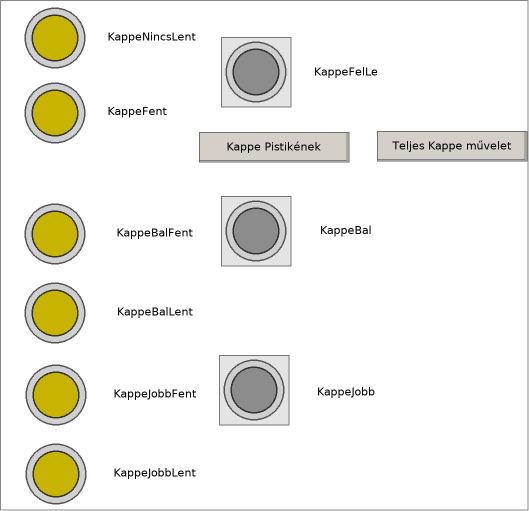
VISUALIZATION TempPistiKappe  // 529x511
    Group (20,3 187x70)
        Lamp1 (0,0 70x70), variable: GVL.bKappepresNincsLegalul, style: Lamp-Lamp1-Yellow
        Label (77,19 110x30), "KappeNincsLent"
    PushSwitch (221,37 70x70), variable: KAPPE.bKappeFelLe, behaviour: TOGGLE, style: Switch-PushSwitch-Gray
    Label (291,57 110x30), "KappeFelLe"
    Lamp1 (20,199 70x70), variable: KAPPE.bKappeBalFent, style: Lamp-Lamp1-Yellow
    Label (100,218 110x30), "KappeBalFent"
    Lamp1 (20,278 70x70), variable: KAPPE.bKappeBalLent, style: Lamp-Lamp1-Yellow
    Label (100,297 110x30), "KappeBalLent"
    PushSwitch (221,196 70x70), variable: KAPPE.bKappeBalFelLe, behaviour: TOGGLE, style: Switch-PushSwitch-Gray
    Label (291,216 110x29), "KappeBal"
    Lamp1 (21,360 70x70), variable: KAPPE.bKappeJobbFent, style: Lamp-Lamp1-Yellow
    Label (100,379 110x30), "KappeJobbFent"
    Lamp1 (21,439 70x70), variable: KAPPE.bKappeJobbLent, style: Lamp-Lamp1-Yellow
    Label (100,458 110x30), "KappeJobbLent"
    PushSwitch (219,355 70x70), variable: KAPPE.bKappeJobbFelLe, behaviour: TOGGLE, style: Switch-PushSwitch-Gray
    Label (291,377 110x30), "KappeJobb"
    Button (199,132 150x30), "Kappe Pistikének", input disabled if: KAPPE.bKappeBalFent<>KAPPE.bKappeJobbFent AND KAPPE.bKappeBalLent<>KAPPE.bKappeJobbLent
        OnMouseUp: execute {
            IF ((KAPPE.bKappeBalFent=TRUE) AND (KAPPE.bKappeBalLent=FALSE) AND (KAPPE.bKappeJobbFent=TRUE) AND (KAPPE.bKappeJobbLent=FALSE)) THEN
            	KAPPE.bKappeBalFelLe:=TRUE;
            	KAPPE.bKappeJobbFelLe:=TRUE;
            ELSE
            	KAPPE.bKappeBalFelLe:=FALSE;
            	KAPPE.bKappeJobbFelLe:=FALSE;
            END_IF
        }
    Button (377,131 150x30), "Teljes Kappe művelet", input disabled if: KAPPE.bKappeBalFent<>KAPPE.bKappeJobbFent AND KAPPE.bKappeBalLent<>KAPPE.bKappeJobbLent
        OnMouseUp: execute { KAPPE.s_InCommand:='START'; }
    Group (20,78 154x70)
        Lamp1 (0,0 70x70), variable: GVL.bKappePresFent, style: Lamp-Lamp1-Yellow
        Label (81,19 73x29), "KappeFent"
END_VISUALIZATION

(* stored: Version 1.1.0.1, ProductVersion 3.1.4024.11
   Visu TempPistiKappe: Id {f31d95ec-78f1-4d20-a515-05560e7c36de} *)
